{attribute 'qualified_only'}
{attribute 'strict'}
TYPE K_Stopper :
(
	ST3K4 := 1, // TMO PPS stopper
    //ST2 := 2
);
END_TYPE

(* stored: Version 1.1.0.1, ProductVersion 3.1.4022.18
   EnumerationTextList K_Stopper: Id {07f71466-4474-4124-a5d9-be5d26954396} *)
